Staubli VAL3: isHome.pgx

program isHome(bool& x_bHome[] (dimensions=1))
begin
  //
  // ask for home status
  //
  x_bHome=cycleStatus:bIsHome
end
